INTERFACE I_Cylinder

METHOD PUBLIC Extend
VAR_INPUT
END_VAR
END_METHOD

METHOD PUBLIC Retract
VAR_INPUT
END_VAR
END_METHOD

END_INTERFACE

(* stored: Version 1.1.0.1, ProductVersion 3.1.4024.4
   Itf I_Cylinder: Id {f0edab36-fb99-4463-90c7-8aca10915ad7}
   Method Extend: Id {7299ce40-6999-4310-94ec-df6856ba424d}
   Method Retract: Id {cf0175fc-f25c-4bb2-a01f-5009985fcaff} *)
